Staubli VAL3: motionSupervisor.pgx

program motionSupervisor()
  local num buffer[8]
  local num value
begin
  while true
    // Sleep until the task enters a runtime error state
    wait(taskStatus(TASK_NAMES["MotionWorker"]) > 1)

    // Clear any invalid pending trajectories
    resetMotion()

    // Notify any clients of the error
    call sendError(1, taskStatus(TASK_NAMES["MotionWorker"]))

    // Resume the task from the next line
    taskResume(TASK_NAMES["MotionWorker"], 1)
  endWhile
end
